(* CODESYS project HelloCODESYS

Project tree, tasks and I/O mapping:
  Device : CODESYS Control Win V3 x64, 3S - Smart Software Solutions GmbH, version 3.5.17.30
    application Application
      libraries: Standard, * (System)
      task MainTask (cyclic, interval t#20ms, priority 1) calls PLC_PRG
      global variables GVL
      program PLC_PRG [ST]
*)

// Device/Application/GVL
{attribute 'qualified_only'}
VAR_GLOBAL
	g_sVar: STRING;
END_VAR

// Device/Application/PLC_PRG
PROGRAM PLC_PRG
VAR
	sVar1: STRING := 'Hello ';
	sVar2: STRING := 'World!';
END_VAR

GVL.g_sVar := CONCAT(sVar1, sVar2);

END_PROGRAM
